# EPICS alarm handler configuration: mps_database/bareTest/alarms/areas/mpln_bc2b_mp01.alhConfig
GROUP NULL MPLN:BC2B:MP01:1
$ALIAS MPS Link Node 62
$GUIDANCE
LTUH MPS
   Group Name: MPLN:BC2B:MP01:1
   Summary PV:  MPLN:BC2B:MP01:1:STATSUMY
$END
CHANNEL  MPLN:BC2B:MP01:1    MPLN:BC2B:MP01:1:MPS_EN_RBV		-----
CHANNEL  MPLN:BC2B:MP01:1    MPLN:BC2B:MP01:1:LC1_MODE_RBV		-----
